	                                                                                                                                                                                                                                                                                                                                                                                                                                                                                                                                                                                                                                                                                                                                                                                                                                                                                                                                                                                                                                                                                                                                                                                                                                                                                                                                                                                                                                                                                                                                                                                                                                                                                                                                                                                                                                                                                                                                                                                                                                                                                                                                                                                                                                                                                                                                                                                                                                                                                                                                                                                                                                                                                                                                                                                                                                                                                                                                                                                                                                                                                                                                                                                                                                                                                                                                                                                                                                                                                                                                                                                                                                                                                                                                                                                                                                                                                                                                                                                                                                                                                                                                                                                                                                                                                                                                                                                                                                                                                                                                                                                                                                                                                                                                                                                                                                                                                                                                                                                                                                                                                                                                                                                                                                                                                                                                                                                                                                                                                                                                                                                                                                                                                                                                                                                                                                                                                                                                                                                                                                                                                                                                                                                                                                                                                                                                                                                                                                                                                                                                                                                                                                                                                                                                                                                                                                                                                                                                                                                                                                                                                                                                                                                                                                                                                                                                                                                                                                                                                                                                                                                                                                                                                                                                                                                                                                                                                                                                                                                                                                                                                                                                                                                                                                                                                                                                                                                                                                                                                                                                                                                                                                                                                                                                                                                                                                                                                                                                                                                                                                                                                                                                                                                                                                                                                                                                                                                                                                                                                                                                                                                                                                                                                                                                                                                                                                                                                                                                                                                                                                                                                                                                                                                                                                                                                                                                                                                                                                                                                                                                                                                                                                                                                                                                                                                                                                                                                                                                                                                                                                                                                                                                                                                                                                                                                                                                                                                                                                                                                                                                                                                                                                                                                                                                                                                                                                                                                                                                                                                                                                                                                                                                                                                                                                                                                                                                                                                                                                                                                                                                                                                                                                                                                                                                                                                                                                                                                                                                                                                                                                                                                                                                                                                                                                                                                                                                                                                                                                                                                                                                                                                                                                                                                                                                                                                                                                                                                                                                                                                                                                                                                                                                                                                                                                                                                                                                                                                                                                                                                                                                                                                                                                                                                                                                                                                                                                                                                                                                                                                                                                                                                                                                                                                                                                                                                                                                                                                                                                                                                                                                                                                                                                                                                                                                                                                                                                                                                                                                                                                                                                                                                                                                                                                                                                                                                                                                                                                                                                                                                                                                                                                                                                                                                                                                                                                                                                                                                                                                                                                                                                                                                                                                                                                                                                                                                                                                                                                                                                                                                                                                                                                                                                                                                                                                                                                                                                                                                                                                                                                                                                                                                                                                                                                                                                                                                                                                                                                                                                                                                                                                                                                                                                                                                                                                                                                                                                                                                                                                                                                                                                                                                                                                                                                                                                                                                                                                                                                                                                                                                                                                                                                                                                                                                                                                                                                                                                                                                                                                                                                                                                                                                                                                                                                                                                                                                                                                                                                                                                                                                                                                                                                                                                                                                                                                                                                                                                                                                                                                                                                                                                                                                                                                                                                                                                                                                                                                                                                                                                                                                                                                                                                                                                                                                                                                                                                                                                                                                                                                                                                                                                                                                                                                                                                                                                                                                                                                                                                                                                                                                                                                                                                                                                                                                                                                                                                                                                                                                                                                                                                                                                                                                                                                                                                                                                                                                                                                                                                                                                                                                                                                                                                                                                                                                                                                                                                                                                                                                                                                                                                                                                                                                                                                                                                                                                                                                                                                                                                                                                                                                                                                                                                                                                                                                                                                                                                                                                                                                                                                                                                                                                                                                                                                                                                                                                                                                                                                                                                                                                                                                                                                                                                                                                                                                                                                                                                                                                                                                                                                                                                                                                                                                                                                                                                                                                                                                                                                                                                                                                                                                                                                                                                                                                                                                                                                                                                                                                                                                                                                                                                                                                                                                                                                                                                                                                                                                                                                                                                                                                                                                                                                                                                                                                                                                                                                                                                                                                                                                                                                                                                                                                                                                                                                                                                                                                                                                                                                                                                                                                                                                                                                                                                                                                                                                                                                                                                                                                                                                                                                                                                                                                                                                                                                                                                                                                                                                                                                                                                                                                                                                                                                                                                                                                                                                                                                                                                                                                                                                                                                                                                                                                                                                                                                                                                                                                                                                                                                                                                                                                                                                                                                                                                                                                                                                                                                                                                                                                                                                                                                                                                                                                                                                                                                                                                                                                                                                                                                                                                                                                                                                                                                                                                                                                                                                                                                                                                                                                                                                                                                                                                                                                                                                                                                                                                                                                                                                                                                                                                                                                                                                                                                                                                                                                                                                                                                                                                                                                                                                                                                                                                                                                                                                                                                                                                                                                                                                                                                                                                                                                                                                                                                                                                                                                                                                                                                                                                                                                                                                                                                                                                                                                                                                                                                                                                                                                                                                                                                                                                                                                                                                                                                                                                                                                                                                                                                                                                                                                                                                                                                                                                                                                                                                                                                                                                                                                                                                                                                                                                                                                                                                                                                                                                                                                                                                                                                                                                                                                                                                                                                                                                                                                                                                                                                                                                                                                                                                                                                                                                                                                                                                                                                                                                                                                                                                                                                                                                                                                                                                                                                                                                                                                                                                                                                                                                                                                                                                                                                                                                                                                                                                                                                                                                                                                                                                                                                                                                                                                                                                                                                                                                                                                                                                                                                                                                                                                                                                                                                                                                                                                                                                                                                                                                                                                                                                                                                                                                                                                                                                                                                                                                                                                                                                                                                                                                                                                                                                                                                                                                                                                                                                                                                                                                                                                                                                                                                                                                                                                                                                                                                                                                                                                                                                                                                                                                                                                                                                                                                                                                                                                                                                                                                                                                                                                                                                                                                                                                                                                                                                                                                                                                                                                                                                                                                                                                                                                                                                                                                                                                                                                                                                                                                                                                                                                                                                                                                                                                                                                                                                                                                                                                                                                                                                                                                                                                                                                                                                                                                                                                                                                                                                                                                                                                                                                                                                                                                                                                                                                                                                                                                                                                                                                                                                                                                                                                                                                                                                                                                                                                                                                                                                                                                                                                                                                                                                                                                                                                                                                                                                                                                                                                                                                                                                                                                                                                                                                                                                                                                                                                                                                                                                                                                                                                                                                                                                                                                                                                                                                                                                                                                                                                                                                                                                                                                                                                                                                                                                                                                                                                                                                                                                                                                                                                                                                                                                                                                                                                                                                                                                                                                                                                                                                                                                                                                                                                                                                                                                                                                                                                                                                                                                                                                                                                                                                                                                                                                                                                                                                                                                                                                                                                                                                                                                                                                                                                                                                                                                                                                                                                                                                                                                                                                                                                                                                                                                                                                                                                                                                                                                                                                                                                                                                                                                                                                                                                                                                                                                                                                                                                                                                                                                                                                                                                                                                                                                                                                                                                                                                                                                                                                                                                                                                                                                                                                                                                                                                                                                                                                                                                                                                                                                                                                                                                                                                                                                                                                                                                                                                                                                                                                                                                                                                                                                                                                                                                                                                                                                                                                                                                                                                                                                                                                                                                                                                                                                                                                                                                                                                                                                                                                                                                                                                                                                                                                                                                                                                                                                                                                                                                                                                                                                                                                                                                                                                                                                                                                                                                                                                                                                                                                                                                                                                                                                                                                                                                                                                                                                                                                                                                                                                                                                                                                                                                                                                                                                                                                                                                                                                                                                                                                                                                                                                                                                                                                                                                                                                                                                                                                                                                                                                                                                                                                                                                                                                                                                                                                                                                                                                                                                                                                                                                                                                                                                                                                                                                                                                                                                                                                                                                                                                                                                                                                                                                                                                                                                                                                                                                                                                                                                                                                                                                                                                                                                                                                                                                                                                                                                                                                                                                                                                                                                                                                                                                                                                                                                                                                                                                                                                                                                                                                                                                                                                                                                                                                                                                                                                                                                                                                                                                                                                                                                                                                                                                                                                                                                                                                                                                                                                                                                                                                                                                                                                                                                                                                                                                                                                                                                                                                                                                                                                                                                                                                                                                                                                                                                                                                                                                                                                                                                                                                                                                                                                                                                                                                                                                                                                                                                                                                                                                                                                                                                                                                                                                                                                                                                                                                                                                                                                                                                                                                                                                                                                                                                                                                                                                                                                                                                                                                                                                                                                                                                                                                                                                                                                                                                                                                                                                                                                                                                                                                                                                                                                                                                                                                                                                                                                                                                                                                                                                                                                                                                                                                                                                                                                                                                                                                                                                                                                                                                                                                                                                                                                                                                                                                                                                                                                                                                                                                                                                                                                                                                                                                                                                                                                                                                                                                                                                                                                                                                                                                                                                                                                                                                                                                                                                                                                                                                                                                                                                                                                                                                                                                                                                                                                                                                                                                                                                                                                                                                                                                                                                                                                                                                                                                                                                                                                                                                                                                                                                                                                                                                                                                                                                                                                                                                                                                                                                                                                                                                                                                                                                                                                                                                                                                                                                                                                                                                                                                                                                                                                                                                                                                                                                                                                                                                                                                                                                                                                                                                                                                                                                                                                                                                                                                                                                                                                                                                                                                                                                                                                                                                                                                                                                                                                                                                                                                                                                                                                                                                                                                                                                                                                                                                                                                                                                                                                                                                                                                                                                                                                                                                                                                                                                                                                                                                                                                                                                                                                                                                                                                                                                                                                                                                                                                                                                                                                                                                                                                                                                                                                                                                                                                                                                                                                                                                                                                                                                                                                                                                                                                                                                                                                                                                                                                                                                                                                                               EW := "EW_LF_CM02.BN04",
	                     Messbereich_Min := "Analogwerte"."LF_CM02.BN04".MB_min,
	                     Messbereich_Max := "Analogwerte"."LF_CM02.BN04".MB_max,
	                     UG_Alarm := "Analogwerte"."LF_CM02.BN04".UG_Alarm,
	                     OG_Alarm := "Analogwerte"."LF_CM02.BN04".OG_Alarm,
	                     GF := "Analogwerte"."LF_CM02.BN04".GF,
	                     Al_Drahtbruch => "Analogwerte"."LF_CM02.BN04".Drahtbruch,
	                     Al_MW_ausserhalb => "Analogwerte"."LF_CM02.BN04".ungueltig,
	                     Messwert := "Panel".IW."LF_CM02.BN04");
	    END_REGION
	
	    REGION Druckmessung
	        // Druck Beutelfiltergehäuse (nach dem Filter)
	        "Analogwert"(Deaktiviert:="DB_Temporaer".Drucksensoren_deaktiviert,
	                     EW := "EW_p_HQ01.BP01",
	                     Messbereich_Min := "Analogwerte"."p_HQ01.BP01".MB_min,
	                     Messbereich_Max := "Analogwerte"."p_HQ01.BP01".MB_max,
	                     UG_Alarm := "Analogwerte"."p_HQ01.BP01".UG_Alarm,
	                     OG_Alarm := "Analogwerte"."p_HQ01.BP01".OG_Alarm,
	                     GF := "Analogwerte"."p_HQ01.BP01".GF,
	                     Al_Drahtbruch => "Analogwerte"."p_HQ01.BP01".Drahtbruch,
	                     Al_MW_ausserhalb => "Analogwerte"."p_HQ01.BP01".ungueltig,
	                     Messwert := #"MW _p_nach Filter_HQ01");
	        // Differenzdruck (vor Filter - nach Filter)
	        "Panel".IW."p_HQ01.BP01" := "Panel".IW."p_CM01.BP03" - #"MW _p_nach Filter_HQ01";
	        
	        // Druck Beutelfiltergehäuse (nach dem Filter)
	        "Analogwert"(Deaktiviert:="DB_Temporaer".Drucksensoren_deaktiviert,
	                     EW := "EW_p_HQ02.BP02",
	                     Messbereich_Min := "Analogwerte"."p_HQ02.BP02".MB_min,
	                     Messbereich_Max := "Analogwerte"."p_HQ02.BP02".MB_max,
	                     UG_Alarm := "Analogwerte"."p_HQ02.BP02".UG_Alarm,
	                     OG_Alarm := "Analogwerte"."p_HQ02.BP02".OG_Alarm,
	                     GF := "Analogwerte"."p_HQ02.BP02".GF,
	                     Al_Drahtbruch => "Analogwerte"."p_HQ02.BP02".Drahtbruch,
	                     Al_MW_ausserhalb => "Analogwerte"."p_HQ02.BP02".ungueltig,
	                     Messwert := #"MW _p_nach Filter_HQ02");
	        // Differenzdruck (vor Filter - nach Filter)
	        "Panel".IW."p_HQ02.BP02" := "Panel".IW."p_CM02.BP06" - #"MW _p_nach Filter_HQ02";
	        
	        // Druck Filterpumpe
	        "Analogwert"(Deaktiviert:="DB_Temporaer".Drucksensoren_deaktiviert,
	                     EW := "EW_p_CM01.BP03",
	                     Messbereich_Min := "Analogwerte"."p_CM01.BP03".MB_min,
	                     Messbereich_Max := "Analogwerte"."p_CM01.BP03".MB_max,
	                     UG_Alarm := "Analogwerte"."p_CM01.BP03".UG_Alarm,
	                     OG_Alarm := "Analogwerte"."p_CM01.BP03".OG_Alarm,
	                     GF := "Analogwerte"."p_CM01.BP03".GF,
	                     Al_Drahtbruch => "Analogwerte"."p_CM01.BP03".Drahtbruch,
	                     Al_MW_ausserhalb => "Analogwerte"."p_CM01.BP03".ungueltig,
	                     Messwert := "Panel".IW."p_CM01.BP03");
	        
	        // Druck Umwälzpumpe
	        "Analogwert"(Deaktiviert:="DB_Temporaer".Drucksensoren_deaktiviert,
	                     EW := "EW_p_CM01.BP04",
	                     Messbereich_Min := "Analogwerte"."p_CM01.BP04".MB_min,
	                     Messbereich_Max := "Analogwerte"."p_CM01.BP04".MB_max,
	                     UG_Alarm := "Analogwerte"."p_CM01.BP04".UG_Alarm,
	                     OG_Alarm := "Analogwerte"."p_CM01.BP04".OG_Alarm,
	                     GF := "Analogwerte"."p_CM01.BP04".GF,
	                     Al_Drahtbruch => "Analogwerte"."p_CM01.BP04".Drahtbruch,
	                     Al_MW_ausserhalb => "Analogwerte"."p_CM01.BP04".ungueltig,
	                     Messwert := "Panel".IW."p_CM01.BP04");
	        // Druck Umwälzpumpe
	        "Analogwert"(Deaktiviert:="DB_Temporaer".Drucksensoren_deaktiviert,
	                     EW := "EW_p_CM03.BP05",
	                     Messbereich_Min := "Analogwerte"."p_CM03.BP05".MB_min,
	                     Messbereich_Max := "Analogwerte"."p_CM03.BP05".MB_max,
	                     UG_Alarm := "Analogwerte"."p_CM03.BP05".UG_Alarm,
	                     OG_Alarm := "Analogwerte"."p_CM03.BP05".OG_Alarm,
	                     GF := "Analogwerte"."p_CM03.BP05".GF,
	                     Al_Drahtbruch => "Analogwerte"."p_CM03.BP05".Drahtbruch,
	                     Al_MW_ausserhalb => "Analogwerte"."p_CM03.BP05".ungueltig,
	                     Messwert := "Panel".IW."p_CM03.BP05");
	        // Druck Filterpumpe
	        "Analogwert"(Deaktiviert:="DB_Temporaer".Drucksensoren_deaktiviert,
	                     EW := "EW_p_CM02.BP06",
	                     Messbereich_Min := "Analogwerte"."p_CM02.BP06".MB_min,
	                     Messbereich_Max := "Analogwerte"."p_CM02.BP06".MB_max,
	                     UG_Alarm := "Analogwerte"."p_CM02.BP06".UG_Alarm,
	                     OG_Alarm := "Analogwerte"."p_CM02.BP06".OG_Alarm,
	                     GF := "Analogwerte"."p_CM02.BP06".GF,
	                     Al_Drahtbruch => "Analogwerte"."p_CM02.BP06".Drahtbruch,
	                     Al_MW_ausserhalb => "Analogwerte"."p_CM02.BP06".ungueltig,
	                     Messwert := "Panel".IW."p_CM02.BP06");
	        
	        // Druck Umwälzpumpe
	        "Analogwert"(Deaktiviert:="DB_Temporaer".Drucksensoren_deaktiviert,
	                     EW := "EW_p_CM02.BP07",
	                     Messbereich_Min := "Analogwerte"."p_CM02.BP07".MB_min,
	                     Messbereich_Max := "Analogwerte"."p_CM02.BP07".MB_max,
	                     UG_Alarm := "Analogwerte"."p_CM02.BP07".UG_Alarm,
	                     OG_Alarm := "Analogwerte"."p_CM02.BP07".OG_Alarm,
	                     GF := "Analogwerte"."p_CM02.BP07".GF,
	                     Al_Drahtbruch => "Analogwerte"."p_CM02.BP07".Drahtbruch,
	                     Al_MW_ausserhalb => "Analogwerte"."p_CM02.BP07".ungueltig,
	                     Messwert := "Panel".IW."p_CM02.BP07");
	        // Druck Umwälzpumpe
	        "Analogwert"(Deaktiviert:="DB_Temporaer".Drucksensoren_deaktiviert,
	                     EW := "EW_p_CM04.BP08",
	                     Messbereich_Min := "Analogwerte"."p_CM04.BP08".MB_min,
	                     Messbereich_Max := "Analogwerte"."p_CM04.BP08".MB_max,
	                     UG_Alarm := "Analogwerte"."p_CM04.BP08".UG_Alarm,
	                     OG_Alarm := "Analogwerte"."p_CM04.BP08".OG_Alarm,
	                     GF := "Analogwerte"."p_CM04.BP08".GF,
	                     Al_Drahtbruch => "Analogwerte"."p_CM04.BP08".Drahtbruch,
	                     Al_MW_ausserhalb => "Analogwerte"."p_CM04.BP08".ungueltig,
	                     Messwert := "Panel".IW."p_CM04.BP08");
	        // Druck Pumpe Entleerung Sammeltank
	        "Analogwert"(Deaktiviert:="DB_Temporaer".Drucksensoren_deaktiviert,
	                     EW := "EW_p_CM05.BP09",
	                     Messbereich_Min := "Analogwerte"."p_CM05.BP09".MB_min,
	                     Messbereich_Max := "Analogwerte"."p_CM05.BP09".MB_max,
	                     UG_Alarm := "Analogwerte"."p_CM05.BP09".UG_Alarm,
	                     OG_Alarm := "Analogwerte"."p_CM05.BP09".OG_Alarm,
	                     GF := "Analogwerte"."p_CM05.BP09".GF,
	                     Al_Drahtbruch => "Analogwerte"."p_CM05.BP09".Drahtbruch,
	                     Al_MW_ausserhalb => "Analogwerte"."p_CM05.BP09".ungueltig,
	                     Messwert := "Panel".IW."p_CM05.BP09");
	    END_REGION
	
	    REGION Durchflussmessung
	        // Durchfluss Versorgung Frischsäure
	        "Analogwert"(Deaktiviert:=FALSE,
	                     EW := "EW_Dfl_GP01.BF01",
	                     Messbereich_Min := "Analogwerte"."Dfl_GP01.BF01".MB_min,
	                     Messbereich_Max := "Analogwerte"."Dfl_GP01.BF01".MB_max,
	                     UG_Alarm := "Analogwerte"."Dfl_GP01.BF01".UG_Alarm,
	                     OG_Alarm := "Analogwerte"."Dfl_GP01.BF01".OG_Alarm,
	                     GF := "Analogwerte"."Dfl_GP01.BF01".GF,
	                     Al_Drahtbruch => "Analogwerte"."Dfl_GP01.BF01".Drahtbruch,
	                     Al_MW_ausserhalb => "Analogwerte"."Dfl_GP01.BF01".ungueltig,
	                     Messwert := "Panel".IW."Dfl_GP01.BF01");
	        // Durchfluss Entsorgung Altsäure
	        "Analogwert"(Deaktiviert:=FALSE,
	                     EW := "EW_Dfl_GP02.BF02",
	                     Messbereich_Min := "Analogwerte"."Dfl_GP02.BF02".MB_min,
	                     Messbereich_Max := "Analogwerte"."Dfl_GP02.BF02".MB_max,
	                     UG_Alarm := "Analogwerte"."Dfl_GP02.BF02".UG_Alarm,
	                     OG_Alarm := "Analogwerte"."Dfl_GP02.BF02".OG_Alarm,
	                     GF := "Analogwerte"."Dfl_GP02.BF02".GF,
	                     Al_Drahtbruch => "Analogwerte"."Dfl_GP02.BF02".Drahtbruch,
	                     Al_MW_ausserhalb => "Analogwerte"."Dfl_GP02.BF02".ungueltig,
	                     Messwert := "Panel".IW."Dfl_GP02.BF02");
	    END_REGION
	    
